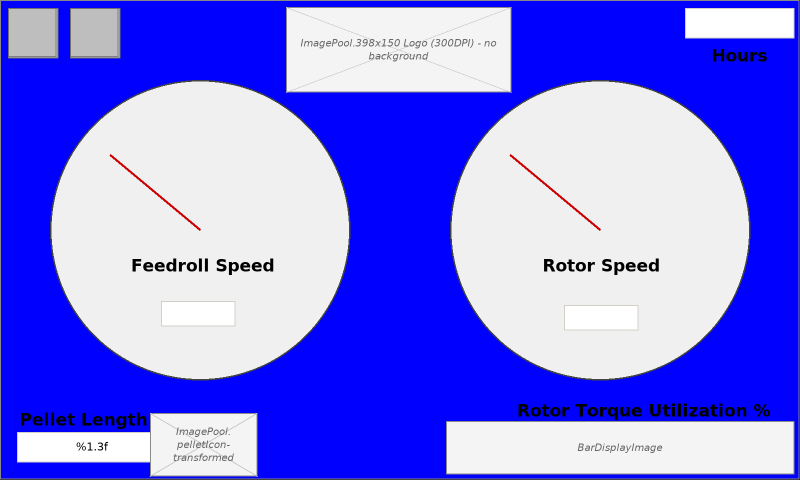
VISUALIZATION Home  // 800x480
    Rectangle (0,0 800x480)
    Meter360 (50,80 300x300), style: Meter-Meter360-Gray, scale format: %.1f, scale 0..100
        p518627256: Ft/Min
    BarDisplayImage (446,421 348x53), value: 0, style: BarDisplayImage-Gray, scale format: %.1f, scale 0..100
    Textfield (17,432 150x30), "%1.3f", text variable: Imperial_Metric_Switching.Pellet_Length_Displayed
    Textfield (161,301 74x25)
    Meter360 (450,80 300x300), style: Meter-Meter360-Gray, scale format: %.1f, scale 0..100
    Textfield (564,305 74x25)
    Image (286,7 225x85), image: ImagePool.398x150 Logo (300DPI) - no background
        OnMouseClick: change screen: Home
    Button (8,8 50x50), tooltip "Login", image: VisuSymbols.Symbols.User
        OnMouseClick: VisuUserMgmt Type=Login
    Label (685,40 109x31), "Hours"
    Textfield (685,8 109x30)
    Label (17,404 133x31), "Pellet Length"
    Label (509,395 270x31), "Rotor Torque Utilization %"
    Label (133,250 140x31), "Feedroll Speed"
    Label (535,250 133x31), "Rotor Speed"
    Button (70,8 50x50), image: VisuSymbols.Symbols.TwoWheels
        OnMouseClick: change screen: Settings_Menu
    Image (150,413 107x63), image: ImagePool.pelletIcon-transformed
        OnMouseClick: OpenDialog Dialog=Preset_Pellet_Length, OpenModal=True, OpenCentered=True
END_VISUALIZATION

(* stored: Version 1.1.0.1, ProductVersion 3.1.4024.12
   Visu Home: Id {8d2acc8d-48b5-4a10-bd97-557a506a34a8} *)
